FUNCTION BETA : REAL
VAR_INPUT
	X : REAL;
	Y : REAL;
END_VAR


(*
version 1.0	26. oct. 2008
programmer 	hugo
tested by		oscat

this function calculates the beta function for real number > 0.

*)

BETA := GAMMA(X) * GAMMA(Y) / GAMMA(x + y);


(* revision history
hm	26. oct. 2008	rev 1.0
	original version

*)

END_FUNCTION

(* stored: Version 1.1.0.1, ProductVersion 3.1.4022.7
   POU BETA: Id {81925f76-62f9-4211-b728-04c6ef48f27b}, SpecialFunc None *)
